PROGRAM MAIN
VAR
END_VAR

END_PROGRAM

(* stored: Version 1.1.0.1
   POU MAIN: Id {63823e6d-fc16-4d7d-b94a-793b0f7de308} *)
